{attribute 'GeneratedUsingTerminal: EJ6224-0000-0016'}
{attribute addProperty BoxType "EJ6224-0000-0016"}
{attribute addProperty Id "DeviceState_InputsDeviceState_Inputs_4751FF764"}
{attribute addProperty CRC "3178000437"}
{attribute addProperty Size "4"}
TYPE Module_2_DeviceState_Inputs_BD6C7035 :
STRUCT
	{attribute addProperty Name "DeviceState_Inputs"}
	DeviceState_Inputs  : DeviceState_Inputs_4751FF76;
END_STRUCT
END_TYPE

(* stored: Version 1.2.0.0, ProductVersion 3.1.4024.9
   DUT Module_2_DeviceState_Inputs_BD6C7035: Id {e04129e1-0a9c-46b2-8f79-0c91de83d7ce} *)
